FUNCTION_BLOCK FB_Izumi
VAR_INPUT
END_VAR
VAR_OUTPUT
	iIzumiInNewton			: INT;	// converted to Newton
END_VAR
VAR
	iIzumiData AT %I* 		: INT;	// measured in mV
	iVoltage AT %I* 		: INT;	// Voltage sensor
END_VAR

iIzumiInNewton 				:= iIzumiData/100;

END_FUNCTION_BLOCK

(* stored: Version 1.1.0.1
   POU FB_Izumi: Id {d432de2a-9cef-45d3-a8f1-b5c1e7f407a3}, SpecialFunc None *)
